(* IEC 61131-3 sources: 89152_FlorisHendrix_AfstudeerProject/89152_FlorisHendrix_ExamenProject/Stations/MachineControl/MachineControl/Class/_CheckOnlineStatus, 1 file *)

(* ---- _CheckOnlineStatus.st ---- *)
(*!
<Class
	Name               = "_CheckOnlineStatus"
	Revision           = "1.4"
	RealtimeTask       = "false"
	CyclicTask         = "true"
	DefCyclictime      = "50 ms"
	BackgroundTask     = "false"
	Sigmatek           = "true"
	OSInterface        = "false"
	HighPriority       = "false"
	Automatic          = "false"
	UpdateMode         = "Prescan"
	SharedCommandTable = "true"
	Objectsize         = "(600,180)"
	Comment            = "class for checking/alarming the online status">
	<Channels>
		<Server Name="Locked" Visualized="false" Initialize="false" WriteProtected="true" Retentive="false" Comment="0 ... communication never was online&#13;&#10;1 ... communication was online"/>
		<Server Name="RestTime" Visualized="false" Initialize="false" WriteProtected="true" Retentive="false" Comment="rest time until alarm will be generated [millisec] (output)"/>
		<Client Name="AlarmCommunication" Required="true" Internal="false" Comment="alarm number for PLC offline alarm (input)"/>
		<Client Name="DelayTime" Required="true" Internal="false" DefValue="20000" Comment="delay time for alarm generating [millisec] (input)"/>
		<Client Name="toTCPComm" Required="true" Internal="false" Comment="Object channel to TCPCommunication."/>
	</Channels>
	<Dependencies>
		<Files>
			<File Path=".\Class\_CheckOnlineStatus\_CheckOnlineStatus_de.pdf"/>
			<File Path=".\Class\_CheckOnlineStatus\_CheckOnlineStatus_en.pdf"/>
		</Files>
	</Dependencies>
	<RevDoku>
		<Owner Company="Sigmatek" Author="FurLuk"/>
		<Dokumentation Revision="1.4" Date="2019-07-09" Author="FurLuk" Company="Sigmatek" Description="Don&apos;t show alarms when the communication is turned off"/>
		<Dokumentation Revision="1.3" Date="2017-01-05" Author="HasHan" Company="Sigmatek" Description="removed the embedded alarmobject to change it for the opmodehandling"/>
		<Dokumentation Revision="1.2" Date="2016-11-04" Author="KaiAnd" Company="Sigmatek" Description="building the locked flag: Wait for first online status AND communication after system start (not only online status)&#13;&#10;also an optional timeDelay is implemented for the alarm generating"/>
		<Dokumentation Revision="1.1" Date="2016-10-10" Author="HubChr" Company="Sigmatek" Description="Added documentation pdfs."/>
		<Dokumentation Revision="1.0" Date="2015-06-24" Company="Sigmatek" Description="Creation."/>
	</RevDoku>
</Class>
*)
_CheckOnlineStatus : CLASS
  //Servers:
	Locked 	: SvrChCmd_DINT;
	RestTime 	: SvrCh_UDINT;
  //Clients:
	toTCPComm 	: CltChCmd_TCPCommunication;
	AlarmCommunication 	: CltCh_DINT;
	DelayTime 	: CltCh_UDINT;
  //Variables:
		TimeMarkAlarm 	: UDINT;
  //Functions:

	FUNCTION VIRTUAL GLOBAL CyWork
		VAR_INPUT
			EAX 	: UDINT;
		END_VAR
		VAR_OUTPUT
			state (EAX) 	: UDINT;
		END_VAR;
  //Tables:
	FUNCTION @STD
		VAR_OUTPUT
			ret_code	: CONFSTATES;
		END_VAR;
	FUNCTION GLOBAL TAB @CT_;
END_CLASS;

#pragma usingLtd TCPCommunication

FUNCTION VIRTUAL GLOBAL _CheckOnlineStatus::CyWork
	VAR_INPUT
		EAX 	: UDINT;
	END_VAR
	VAR_OUTPUT
		state (EAX) 	: UDINT;
	END_VAR
  VAR
  	myOnlineWarning : DINT;
  	myOnlineAlarm   : DINT;
  END_VAR

  //-----------------------------------------------------------------
  //  INIT
  //-----------------------------------------------------------------
  DelayTime := DelayTime.Read();
  myOnlineWarning := 0;
  myOnlineAlarm   := 0;

  // v1.4 -- FurLuk -- don't show CommunicationError if Communication is disabled
  if (toTCPComm.DeactivateCom = 0) then

    //-----------------------------------------------------------------
    //  Online-Alarm:
    //-----------------------------------------------------------------

    // online and communication ... Status OK!
    if ( (toTCPComm.Online <> 0) &
         (toTCPComm.TransferRateReceive <> 0) ) then
      Locked := 1;      // Communication was online after system start

  //  elsif (locked = 1) then
    else
      myOnlineWarning := 1;
    end_if;

    //-----------------------------------------------------------------
    //  building the alarm with delayTimer
    //-----------------------------------------------------------------

    // no online warning
    if (myOnlineWarning = 0) then
      TimeMarkAlarm := ops.tAbsolute;

    // online warning!
    else
      // time delay
      if ((ops.tAbsolute - TimeMarkAlarm) >= DelayTime) then

        myOnlineAlarm := 1;   // set alarm
      end_if;
    end_if;

    // write status to alarm server
    if (AlarmCommunication.Read() <> myOnlineAlarm) then
      AlarmCommunication.Write(input:=myOnlineAlarm);
    end_if;

    // write rest time to server
    RestTime := DelayTime - (ops.tAbsolute - TimeMarkAlarm);
    if (RestTime$DINT < 0) then
      RestTime := 0;
    end_if;

    //-----------------------------------------------------------------
  else

    // v1.4 -- FurLuk -- be able to reset an alarm that accured bevor turned off,
    // or if not turned off at the same time
    if (myOnlineAlarm <> AlarmCommunication.Read()) then
      AlarmCommunication.Write(input:=myOnlineAlarm);
    end_if;

  end_if;

	state := READY;

END_FUNCTION
